(* IEC 61131-3 sources: programs/VI-54/VI-54_20171205/VI-54_20171205/Stations/Screen/LseClass170718/Class/EventExport, 1 file *)

(* ---- EventExport.st ---- *)
(*!
<Class
	Name               = "EventExport"
	Revision           = "1.1"
	RealtimeTask       = "false"
	CyclicTask         = "false"
	BackgroundTask     = "true"
	DefBackground      = "10 ms"
	Sigmatek           = "false"
	OSInterface        = "false"
	HighPriority       = "false"
	Automatic          = "false"
	UpdateMode         = "Prescan"
	SharedCommandTable = "true"
	Objectsize         = "(540,180)"
	Comment            = "class for starting the event export of the EventJournal">
	<Channels>
		<Server Name="ClassSvr" Visualized="false" Initialize="false" WriteProtected="true" Retentive="false" Comment="class server"/>
		<Server Name="ExFilt_Date1" Visualized="true" Initialize="false" WriteProtected="false" Retentive="false" Comment="begin-date for export"/>
		<Server Name="ExFilt_Date2" Visualized="true" Initialize="false" WriteProtected="false" Retentive="false" Comment="end-date for export"/>
		<Server Name="ExportFilter" Visualized="true" Initialize="true" DefValue="2#1111111111" WriteProtected="false" Retentive="false" Comment="Filter for exporting the event types&#13;&#10;Bit 0 = System Messsage Cat.1&#13;&#10;Bit 1 = System Messsage Cat.2&#13;&#10;Bit 2 = System Messsage Cat.3&#13;&#10;Bit 3 = System Messsage Cat.4&#13;&#10;Bit 4 = Alarm&#13;&#10;Bit 5 = System On/Off&#13;&#10;Bit 6 = Login/Logout&#13;&#10;Bit 7 = value changes&#13;&#10;Bit 8 = User-Event&#13;&#10;Bit 9 = switching operation mode"/>
		<Server Name="StartExport" Visualized="true" Initialize="false" WriteProtected="false" Retentive="false" Comment="1 = start-command for exporting events from EventJournal"/>
		<Client Name="coEventJournal" Required="true" Internal="false" Comment="object channel to EventJournal"/>
	</Channels>
	<RevDoku>
		<Owner Company="Sigmatek"/>
		<Dokumentation Revision="1.1" Date="2016-06-15" Author="KaiAnd" Company="Sigmatek" Description="export filter included"/>
		<Dokumentation Revision="1.0" Date="2015-09-22" Company="Sigmatek" Description="Creation."/>
	</RevDoku>
</Class>
*)
EventExport : CLASS
	TYPE
	  T_BITS : BDINT  //! <Type Public="true" Name="T_BITS"/>
	  [
	    1 Bit1,
	    2 Bit2,
	    3 Bit3,
	    4 Bit4,
	    5 Bit5,
	    6 Bit6,
	    7 Bit7,
	    8 Bit8,
	    9 Bit9,
	    10 Bit10,
	    11 Bit11,
	    12 Bit12,
	    13 Bit13,
	    14 Bit14,
	    15 Bit15,
	    16 Bit16,
	    17 Bit17,
	    18 Bit18,
	    19 Bit19,
	    20 Bit20,
	    21 Bit21,
	    22 Bit22,
	    23 Bit23,
	    24 Bit24,
	    25 Bit25,
	    26 Bit26,
	    27 Bit27,
	    28 Bit28,
	    29 Bit29,
	    30 Bit30,
	    31 Bit31,
	    32 Bit32,
	  ];
	END_TYPE
  //Servers:
	ClassSvr 	: SvrChCmd_DINT;
	StartExport 	: SvrCh_DINT;
	ExportFilter 	: SvrCh_T_BITS_PTofCls_EventExport;
	ExFilt_Date1 	: SvrCh_HDINT;
	ExFilt_Date2 	: SvrCh_HDINT;
  //Clients:
	coEventJournal 	: CltChCmd_EventJournal;
  //Variables:
  //Functions:

	FUNCTION VIRTUAL GLOBAL Init;

	FUNCTION VIRTUAL GLOBAL Background
		VAR_INPUT
			EAX 	: UDINT;
		END_VAR
		VAR_OUTPUT
			state (EAX) 	: UDINT;
		END_VAR;

	FUNCTION VIRTUAL GLOBAL ExportFilter::Write
		VAR_INPUT
			input (EAX) 	: EventExport::T_BITS;
		END_VAR
		VAR_OUTPUT
			result (EAX) 	: EventExport::T_BITS;
		END_VAR;
  //Tables:
	FUNCTION @STD
		VAR_OUTPUT
			ret_code	: CONFSTATES;
		END_VAR;
	FUNCTION GLOBAL TAB @CT_;
END_CLASS;

#pragma usingLtd EventJournal

FUNCTION VIRTUAL GLOBAL EventExport::Init

    // check the inputs
    if (ExFilt_Date1 = 0) then
      ExFilt_Date1 := 16#07D11011;  // 01.01.2001
      ExFilt_Date1.Write(input:=ExFilt_Date1);
    end_if;
    if (ExFilt_Date2 = 0) then
      ExFilt_Date2 := 16#08331014;  // 01.01.2099
      ExFilt_Date2.Write(input:=ExFilt_Date2);
    end_if;

END_FUNCTION

FUNCTION VIRTUAL GLOBAL EventExport::Background
	VAR_INPUT
		EAX 	: UDINT;
	END_VAR
	VAR_OUTPUT
		state (EAX) 	: UDINT;
	END_VAR

  if (StartExport = 1) then

    // check the inputs
    if (ExFilt_Date1 = 0) then
      ExFilt_Date1 := 16#07D11011;  // 01.01.2001
      ExFilt_Date1.Write(input:=ExFilt_Date1);
    end_if;
    if (ExFilt_Date2 = 0) then
      ExFilt_Date2 := 16#08331014;  // 01.01.2099
      ExFilt_Date2.Write(input:=ExFilt_Date2);
    end_if;

    // start export
    case  coEventJournal.ExportEvents(ExportFilter:=ExportFilter,
                                      ExFilt_Date1:=ExFilt_Date1, ExFilt_Date2:=ExFilt_Date2,
                                      ExFilt_Time1:=0, ExFilt_Time2:=16#FFffFFff)  of
      // Export fertig
      READY:
        StartExport := 0;

      // Export in arbeit
      BUSY:

      // Export mit Error abgebrochen
      ERROR:
        StartExport := 0;

    end_case;

  end_if;

	state := READY;

END_FUNCTION

FUNCTION VIRTUAL GLOBAL EventExport::ExportFilter::Write
	VAR_INPUT
		input (EAX) 	: EventExport::T_BITS;
	END_VAR
	VAR_OUTPUT
		result (EAX) 	: EventExport::T_BITS;
	END_VAR
  VAR
    mydat : UDINT;
	  para  : UDINT;
  END_VAR

  mydat := ExportFilter$UDINT;
  para  := input$UDINT;

  if(para and 16#80000000) then
    if(para = 16#80000000) then
	    mydat := mydat or 16#80000000;
	  else
      mydat := mydat or (para and 16#7FFFFFFF);
    end_if;
  else
    if(para = 0) then
      mydat := mydat and 16#7FFFFFFF;
    else
	  mydat := mydat and (16#FFFFFFFF xor para);
	  end_if;
  end_if;

  result       := mydat;
  ExportFilter := mydat;

END_FUNCTION
